// TIA Portal project "CODE_2" (V16)

(* hardware
DEVICE "S7-1200 station_1"  S7-1200 Station
   slot 0: "Rack_0"  S7-1200 Rack  Rack  V1.0
   slot 1: "PLC_1"  CPU 1212C DC/DC/DC  6ES7 212-1AE40-0XB0  V4.1
   slot 2: "AI 4x13BIT_1"  6ES7 231-4HD32-0XB0  V2.1
DEVICE "PC-System_1"  SIMATIC PC station
   slot 0: "SIMATIC PC station"  Rail  SIMATIC PC-Station  V1.0
      slot 125: "Stationmanager"  Station_Manager  V6.0.4
   slot 1: "HMI_RT_1"  WinCC RT Advanced  6AV2 104-0xxxx-xxxx  16.0.0.0
      slot 33792: "Computer interface"  Host interface
   slot 2: "IE general_1"  IE General  IE_CP  V8.2.0
*)

// ===== PLC "PLC_1"  CPU 1212C DC/DC/DC =====

VAR_GLOBAL   // PLC tag table "Default tag table"
   "System_Byte" AT %MB100 : Byte;
   "FirstScan" AT %M100.0 : Bool;
   "DiagStatusUpdate" AT %M100.1 : Bool;
   "AlwaysTRUE" AT %M100.2 : Bool;
   "AlwaysFALSE" AT %M100.3 : Bool;
   "Clock_Byte" AT %MB101 : Byte;
   "Clock_10Hz" AT %M101.0 : Bool;
   "Clock_5Hz" AT %M101.1 : Bool;
   "Clock_2.5Hz" AT %M101.2 : Bool;
   "Clock_2Hz" AT %M101.3 : Bool;
   "Clock_1.25Hz" AT %M101.4 : Bool;
   "Clock_1Hz" AT %M101.5 : Bool;
   "Clock_0.625Hz" AT %M101.6 : Bool;
   "Clock_0.5Hz" AT %M101.7 : Bool;
   "START" AT %M0.1 : Bool;
   "STOP" AT %M0.2 : Bool;
   "RESET" AT %M0.3 : Bool;
   "EMER" AT %M0.4 : Bool;
   "PUMP1" AT %Q0.0 : Bool;
   "PUMP2" AT %Q0.1 : Bool;
   "PUMP3" AT %Q0.2 : Bool;
   "RUN_L" AT %Q0.3 : Bool;
   "STOP_L" AT %Q0.4 : Bool;
   "ERROR_L" AT %Q0.5 : Bool;
   "PRESSURE" AT %MD20 : Real;
   "Tag" AT %MD24 : Real;
   "AI0" AT %MW96 : Word;
END_VAR

DATA_BLOCK "SCL"   // DB1
{ S7_Optimized_Access := 'TRUE' }
VERSION : 0.1
   VAR
      TT : Int;
      TIMER0 : TON_TIME;
      TIMER1 : TON_TIME;
      TIMER2 : TON_TIME;
      TIMER3 : TON_TIME;
      TIMER4 : TON_TIME;
      TIMER5 : TON_TIME;
      TIMER6 : TON_TIME;
      TIMER7 : TON_TIME;
      TIMER_30 : TON_TIME;
   END_VAR
BEGIN
END_DATA_BLOCK

ORGANIZATION_BLOCK "Main"   // OB1, LAD, ProgramCycle
TITLE = "Main Program Sweep (Cycle)"
{ S7_Optimized_Access := 'TRUE' }
VERSION : 0.1
   VAR_INPUT
      Initial_Call : Bool;   // Initial call of this OB
      Remanence : Bool;   // =True, if remanent data are available
   END_VAR
BEGIN

REGION Network 1 (SCL)
   REGION ĐỌC TÍN HIỆU ANALOG
       "PRESSURE" := SCALE_X(MIN := 0,
                             VALUE := NORM_X(MIN := 0, VALUE := "AI0", MAX := 27648),
                             MAX := 87);
   END_REGION ;

   IF "FirstScan" = 1 THEN
       "SCL".TT := 0;
   END_IF;

   CASE "SCL".TT OF
       0:
           REGION TRẠNG THÁI BAN ĐẦU
               "STOP_L" := TRUE;
               "RUN_L" := FALSE;
               "PUMP1" := FALSE;
               "PUMP2" := FALSE;
               "PUMP3" := FALSE;
               REGION NÚT NHẤN START
                   IF "START" = 1 THEN
                       "SCL".TT := 1;
                   END_IF;
               END_REGION
           END_REGION
           ;
       1:
           REGION TRẠNG THÁI BÌNH THƯỜNG
               "STOP_L" := 0;
               "RUN_L" := 1;
               REGION P<30                
                   IF "PRESSURE" < 30 THEN
                       //Bật 1 bơm sau mỗi 5 phút nếu P<30
                       "SCL".TIMER0(IN := ((NOT "PUMP1" & NOT "PUMP2" & NOT "PUMP3") OR ("PUMP1" & NOT "PUMP2" & NOT "PUMP3") OR ("PUMP1" & NOT "PUMP2" & "PUMP3")) & "PRESSURE" < 30,
                                    PT := T#10s);
                       "SCL".TIMER1(IN := "PUMP1" & "PUMP2" & NOT "PUMP3" & "PRESSURE" < 30,
                                    PT := T#10s);
                       "SCL".TIMER2(IN := "PUMP1" & "PUMP2" & "PUMP3" & "PRESSURE" < 30,
                                    PT := T#10s);
                       "SCL".TIMER3(IN := (NOT "PUMP1" & NOT "PUMP2" & "PUMP3") OR (NOT "PUMP1" & "PUMP2" & "PUMP3") OR (NOT "PUMP1" & "PUMP2" & NOT "PUMP3"),
                                    PT := T#10s);
                       RESET_TIMER("SCL".TIMER_30);
                       IF (NOT "PUMP1" & NOT "PUMP2" & NOT "PUMP3" ) OR ((NOT"PUMP1" & NOT "PUMP2" & "PUMP3") OR (NOT "PUMP1" & "PUMP2" & "PUMP3") OR (NOT "PUMP1" & "PUMP2" & NOT "PUMP3")) & "SCL".TIMER3.Q THEN
                           "PUMP1" := TRUE;
                       ELSIF (("PUMP1" & NOT "PUMP2" & NOT "PUMP3") OR ("PUMP1" & NOT "PUMP2" & "PUMP3")) & "SCL".TIMER0.Q THEN
                           "PUMP2" := TRUE;
                           RESET_TIMER("SCL".TIMER0);
                       ELSIF ("PUMP1" & "PUMP2" & NOT "PUMP3" & "SCL".TIMER1.Q) THEN
                           "PUMP3" := TRUE;
                           RESET_TIMER("SCL".TIMER1);
                       END_IF;
                   END_IF;
               END_REGION

               REGION 30<=P<=50 
                   //Giữ nguyên trạng thái
                   IF "PRESSURE" >= 30 & "PRESSURE" <= 50 THEN
                       RESET_TIMER("SCL".TIMER0);
                       RESET_TIMER("SCL".TIMER1);
                       RESET_TIMER("SCL".TIMER2);
                   END_IF;
               END_REGION

               REGION P>50
                   //Tắt 1 bơm sau mỗi 5 phút nếu P>50
                   "SCL".TIMER4(IN := (("PUMP1" & "PUMP2" & "PUMP3") OR ("PUMP1" & NOT "PUMP2" & NOT "PUMP3") OR ("PUMP1" & "PUMP2" & NOT "PUMP3") OR ("PUMP1" & NOT "PUMP2" & "PUMP3")) & "PRESSURE" > 50,
                                PT := T#10s);
                   "SCL".TIMER5(IN := (NOT "PUMP1" & "PUMP2" & "PUMP3") & "PRESSURE" > 50,
                                PT := T#10s);
                   "SCL".TIMER6(IN := ((NOT "PUMP1" & NOT "PUMP2" & "PUMP3") OR (NOT "PUMP1" & "PUMP2" & NOT "PUMP3")) & "PRESSURE" > 50,
                                PT := T#10s);
                   "SCL".TIMER_30(IN := NOT "PUMP1" & NOT "PUMP2" & NOT "PUMP3" & "PRESSURE" > 50 & "PRESSURE" < 60,
                                  PT := T#30s);
                   IF "PRESSURE" > 50 THEN
                       RESET_TIMER("SCL".TIMER2);
                       IF (("PUMP1" & "PUMP2" & "PUMP3") OR ("PUMP1" & NOT "PUMP2" & NOT "PUMP3") OR ("PUMP1" & "PUMP2" & NOT "PUMP3") OR ("PUMP1" & NOT "PUMP2" & "PUMP3")) & "SCL".TIMER4.Q THEN
                           "PUMP1" := FALSE;
                           RESET_TIMER("SCL".TIMER4);
                       ELSIF (NOT "PUMP1" & "PUMP2" & "PUMP3" & "SCL".TIMER5.Q) THEN
                           "PUMP1" := FALSE;
                           "PUMP2" := FALSE;
                           RESET_TIMER("SCL".TIMER5);
                       ELSIF (NOT "PUMP1" & NOT "PUMP2" & "PUMP3" & "SCL".TIMER6.Q) OR (NOT "PUMP1" & "PUMP2" & NOT "PUMP3" & "SCL".TIMER6.Q) THEN
                           "PUMP1" := FALSE;
                           "PUMP2" := FALSE;
                           "PUMP3" := FALSE;
                           RESET_TIMER("SCL".TIMER6);
                       END_IF;
                   END_IF;
               END_REGION

               REGION TRẠNG THÁI BỊ LỖI
                   IF "SCL".TIMER2.Q OR "SCL".TIMER_30.Q OR "PRESSURE" > 60 THEN
                       "SCL".TT := 2;
                   END_IF;
               END_REGION

               REGION NÚT NHẤN STOP
                   IF "STOP" THEN
                       RESET_TIMER("SCL".TIMER0);
                       RESET_TIMER("SCL".TIMER1);
                       RESET_TIMER("SCL".TIMER2);
                       "SCL".TT := 0;
                   END_IF;
               END_REGION

               REGION NÚT NHẤN EMERGENCY
                   IF "EMER" THEN
                       "SCL".TT := 3;
                   END_IF;
               END_REGION
           END_REGION
           ;
       2:
           REGION TRƯỜNG HỢP LỖI
               "ERROR_L" := TRUE;
               "STOP_L" := FALSE;
               "RUN_L" := FALSE;
               "PUMP1" := FALSE;
               "PUMP2" := FALSE;
               "PUMP3" := FALSE;
               REGION RESET LỖI
                   IF "RESET" THEN
                       "ERROR_L" := FALSE;
                       "SCL".TT := 0;
                       RESET_TIMER("SCL".TIMER0);
                       RESET_TIMER("SCL".TIMER1);
                       RESET_TIMER("SCL".TIMER2);
                       RESET_TIMER("SCL".TIMER_30);
                   END_IF;
               END_REGION

           END_REGION
           ;
       3: 
           REGION TRƯỜNG HỢP KHẨN CẤP
               "RUN_L" := FALSE;
               "STOP_L" := TRUE;
               "ERROR_L" := TRUE;
               "PUMP1" := FALSE;
               "PUMP2" := FALSE;
               "PUMP3" := FALSE;
               REGION RESET TRƯỜNG HỢP KHẨN CẤP
                   IF "RESET" THEN
                       "ERROR_L" := FALSE;
                       "SCL".TT := 0;
                       RESET_TIMER("SCL".TIMER0);
                       RESET_TIMER("SCL".TIMER1);
                       RESET_TIMER("SCL".TIMER2);
                       RESET_TIMER("SCL".TIMER_30);
                   END_IF;
               END_REGION

           END_REGION
           ;
   END_CASE;
END_REGION
END_ORGANIZATION_BLOCK

(* ===== HMI "HMI_RT_1" =====
system functions are stored by id; their names below are inferred from use
connection "HMI_Connection_1": ETHERNET, S7_1200_OMS
connection "HMI_Connection_2": ETHERNET, S7_1200_OMS

HMI tags "Default tag table"
   "RUN_L" : Bool = PLC RUN_L AT %Q0.3, 100 ms
   "STOP_L" : Bool = PLC STOP_L AT %Q0.4, 100 ms
   "START" : Bool = PLC START AT %M0.1, 100 ms
   "PUMP1" : Bool = PLC PUMP1 AT %Q0.0, 100 ms
   "PUMP2" : Bool = PLC PUMP2 AT %Q0.1, 100 ms
   "PUMP3" : Bool = PLC PUMP3 AT %Q0.2, 100 ms
   "PRESSURE" : Real = PLC PRESSURE AT %MD20, 100 ms
   "STOP" : Bool = PLC STOP AT %M0.2, 100 ms
   "RESET" : Bool = PLC RESET AT %M0.3, 100 ms
   "EMER" : Bool = PLC EMER AT %M0.4, 100 ms
   "ERROR_L" : Bool = PLC ERROR_L AT %Q0.5, 100 ms
   "AI0" : Word = PLC AI0 AT %MW96, 100 ms

screen "Screen_1" 1024x768
   Button "Button_1" at 395,551 size 96x32; TextOff 'START'
      Appearance <- "START"
      on Press: SetBit("START")
      on Release: ResetBit("START")
   Circle "Circle_1" at 537,544 size 39x39
      Appearance <- "RUN_L"
   Circle "Circle_2" at 537,616 size 39x39
      Appearance <- "STOP_L"
   Button "Button_2" at 395,600 size 96x32; TextOff 'STOP'
      on Release: ResetBit("STOP")
      on Press: SetBit("STOP")
      Appearance <- "STOP"
   Button "Button_3" at 395,649 size 96x32; TextOff 'RESET'
      on Release: ResetBit("RESET")
      on Press: SetBit("RESET")
      Appearance <- "RESET"
   Button "Button_4" at 395,699 size 96x32; TextOff 'EMER'
      on Release: ResetBit("EMER")
      Appearance <- "EMER"
      on Press: SetBit("EMER")
   Circle "Circle_6" at 537,685 size 39x39
      Appearance <- "ERROR_L"
   SymbolLibrary "Symbol library_1" at 40,489 size 51x73
      Appearance <- "PUMP1"
   SymbolLibrary "Symbol library_3" at 74,218 size 12x271
      Appearance <- "PUMP1"
   SymbolLibrary "Symbol library_2" at 110,489 size 51x73
      Appearance <- "PUMP2"
   SymbolLibrary "Symbol library_4" at 180,489 size 51x73
      Appearance <- "PUMP3"
   SymbolLibrary "Symbol library_8" at 144,217 size 12x272
      Appearance <- "PUMP2"
   SymbolLibrary "Symbol library_9" at 215,220 size 12x269
      Appearance <- "PUMP3"
   SymbolLibrary "Symbol library_11" at 135,196 size 29x26
      Appearance <- "RUN_L"
   SymbolLibrary "Symbol library_13" at 100,197 size 37x12
      Appearance <- "RUN_L"
   SymbolLibrary "Symbol library_14" at 162,197 size 44x12
      Appearance <- "RUN_L"
   SymbolLibrary "Symbol library_15" at 206,196 size 29x26
      Appearance <- "RUN_L"
   SymbolLibrary "Symbol library_16" at 234,197 size 446x12
      Appearance <- "RUN_L"
   SymbolLibrary "Symbol library_18" at 359,144 size 47x61
   SymbolLibrary "Symbol library_19" at 419,147 size 38x54
      ProcessValue <- "PRESSURE"
   TextField "Text field_6" at 570,142 size 39x35; Text 'psi'
   GraphicView "Graphic view_3" at 8,557 size 259x190; Picture "Graphic_11"
   TextField "Text field_2" at 538,584 size 37x21; Text 'RUN'
   TextField "Text field_4" at 536,655 size 42x21; Text 'STOP'
   TextField "Text field_5" at 529,723 size 55x21; Text 'ERROR'
   TextField "Text field_3" at 402,500 size 166x29; Text 'Bảng điều khiển'
   GraphicView "Graphic view_8" at 724,616 size 112x141; Picture "Graphic_7"
   GraphicView "Graphic view_2" at 757,595 size 267x173; Picture "Graphic_8"
   GraphicView "Graphic view_4" at 670,427 size 66x103; Picture "Graphic_9"
   TextField "Text field_1" at 356,13 size 348x33; Text 'ĐỒ ÁN HỌC PHẦN TỰ ĐỘNG'
   TextField "Text field_7" at 304,62 size 442x42; Text 'SỬ DỤNG NGÔN NGỮ SCL VIẾT CHƯƠNG TRÌNH ĐIỀU KHIỂN HỆ THỐNG BƠM ĐIỀU ÁP TÒA NHÀ'
   TextField "Text field_8" at 11,468 size 55x21; Text 'BƠM 1'
   TextField "Text field_9" at 90,468 size 55x21; Text 'BƠM 2'
   TextField "Text field_10" at 160,468 size 55x21; Text 'BƠM 3'
   Slider "Slider_1" at 438,222 size 92x260; Caption 'SIMATIC'
      ProcessValue <- "AI0"
   IOField "I/O field_1" at 471,150 size 96x32; FormatPattern 99.9
      ProcessValue <- "PRESSURE"
   SymbolLibrary "Symbol library_7" at 675,167 size 61x46
   SymbolLibrary "Symbol library_6" at 732,100 size 243x430
   SymbolLibrary "Symbol library_5" at 71,196 size 29x26
      Appearance <- "RUN_L"
*)